FUNCTION_BLOCK TEST_LEN (* Test LE functions of numerical values *)
  (* Standard: IEC 61499-1 *)
  (* Version 0.0, 2006-09-11, JHC, Holobloc Inc *)
  (* Compiler header: package fb.rt.test; *)
  (* Compiler classdef: SimpleFB *)
  (* Compiler Java Sun JDK 1.5.0 *)
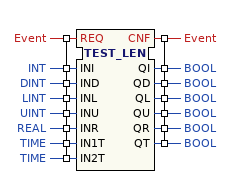
  EVENT_INPUT
    REQ WITH INI, INL, INU, IND, INR, IN1T, IN2T;
  END_EVENT
  EVENT_OUTPUT
    CNF WITH QI, QD, QL, QU, QR, QT;
  END_EVENT
  VAR_INPUT
    INI : INT;
    IND : DINT;
    INL : LINT;
    INU : UINT;
    INR : REAL;
    IN1T : TIME;
    IN2T : TIME;
  END_VAR
  VAR_OUTPUT
    QI : BOOL;
    QD : BOOL;
    QL : BOOL;
    QU : BOOL;
    QR : BOOL;
    QT : BOOL;
  END_VAR
  ALGORITHM REQ IN FBD:
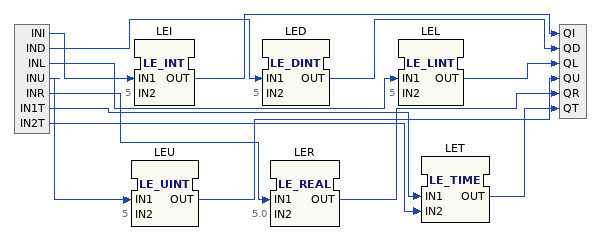
    FBS
      LEI : LE_INT(IN2 := 5);
      LED : LE_DINT(IN2 := 5);
      LEL : LE_LINT(IN2 := 5);
      LEU : LE_UINT(IN2 := 5);
      LER : LE_REAL(IN2 := 5.0);
      LET : LE_TIME;
    END_FBS
    DATA_CONNECTIONS
      INI TO LEI.IN1;
      IND TO LED.IN1;
      INL TO LEL.IN1;
      INU TO LEU.IN1;
      INR TO LER.IN1;
      LEI.OUT TO QI;
      LED.OUT TO QD;
      LEL.OUT TO QL;
      LEU.OUT TO QU;
      LER.OUT TO QR;
      LET.OUT TO QT;
      IN1T TO LET.IN1;
      IN2T TO LET.IN2;
    END_CONNECTIONS
  END_ALGORITHM
END_FUNCTION_BLOCK
